{attribute 'linkalways'} 
{attribute 'no_explicit_call' := 'This FB is a CLASS and must be accessed using methods or properties'}
{attribute 'enable_dynamic_creation'}
FUNCTION_BLOCK _TcVnKeyPoint EXTENDS StructuredDatatypeBase
VAR
	localData : TcVnKeyPoint;
	activeData : REFERENCE TO TcVnKeyPoint REF= localData;
    _aPoint : _TcVnPoint2_REAL();
    _fDiameter : _REAL(localdata.fDiameter);
    _fAngle : _REAL(localdata.fAngle);
    _fResponse : _REAL(localdata.fResponse);
    _nOctave : _DINT(localdata.nOctave);
    _nClassId : _DINT(localdata.nClassId);
END_VAR

PROPERTY PUBLIC Address : PVOID
GET
Address := ADR(activeData);
END_GET
END_PROPERTY

PROPERTY PUBLIC aPoint : REFERENCE TO _TcVnPoint2_REAL
GET
aPoint REF= _aPoint;
END_GET
END_PROPERTY

METHOD PUBLIC ClearReference
VAR_INPUT
END_VAR
activeData REF= localData;
SetMemberReference();
END_METHOD

METHOD PUBLIC Clone : I_Datatype
VAR
    pClone : POINTER TO _TcVnKeyPoint;
END_VAR
pClone := __NEW(_TcVnKeyPoint());
pClone^.Value := Value;
Clone := pClone^;
END_METHOD

PROPERTY PUBLIC fAngle : REFERENCE TO _REAL
GET
fAngle REF= _fAngle;
END_GET
END_PROPERTY

METHOD FB_init : BOOL
VAR_INPUT
	bInitRetains : BOOL; // if TRUE, the retain variables are initialized (warm start / cold start)
	bInCopyCode : BOOL;  // if TRUE, the instance afterwards gets moved into the copy code (online change)
END_VAR
SetMemberReference();
AddMember('aPoint', _aPoint);
AddMember('fDiameter', _fDiameter);
AddMember('fAngle', _fAngle);
AddMember('fResponse', _fResponse);
AddMember('nOctave', _nOctave);
AddMember('nClassId', _nClassId);
END_METHOD

PROPERTY PUBLIC fDiameter : REFERENCE TO _REAL
GET
fDiameter REF= _fDiameter;
END_GET
END_PROPERTY

PROPERTY PUBLIC fResponse : REFERENCE TO _REAL
GET
fResponse REF= _fResponse;
END_GET
END_PROPERTY

PROPERTY PUBLIC Identifier : T_MAXSTRING
GET
Identifier := 'TcVnKeyPoint';
END_GET
END_PROPERTY

METHOD PUBLIC MakeReferenceTo
VAR_INPUT
	ReferenceTarget : REFERENCE TO TcVnKeyPoint;
END_VAR
activeData REF= ReferenceTarget;
SetMemberReference();
END_METHOD

PROPERTY PUBLIC nClassId : REFERENCE TO _DINT
GET
nClassId REF= _nClassId;
END_GET
END_PROPERTY

PROPERTY PUBLIC nOctave : REFERENCE TO _DINT
GET
nOctave REF= _nOctave;
END_GET
END_PROPERTY

METHOD PROTECTED SetMemberReference
VAR_INPUT
END_VAR
_aPoint.MakeReferenceTo(activeData.aPoint);
_fDiameter.MakeReferenceTo(activeData.fDiameter);
_fAngle.MakeReferenceTo(activeData.fAngle);
_fResponse.MakeReferenceTo(activeData.fResponse);
_nOctave.MakeReferenceTo(activeData.nOctave);
_nClassId.MakeReferenceTo(activeData.nClassId);
END_METHOD

PROPERTY PUBLIC Size : UDINT
GET
Size := SIZEOF(activeData);
END_GET
END_PROPERTY

METHOD TryMakeReferenceTo : BOOL
VAR_INPUT
	Target : I_Datatype;
END_VAR
VAR
	pTargetData : POINTER TO TcVnKeyPoint;
END_VAR
IF NOT IsEquivalentTo(Target) THEN
	RETURN;
END_IF

pTargetData := Target.Address;
activeData REF= pTargetData^;
SetMemberReference();
TryMakeReferenceTo := TRUE;
END_METHOD

PROPERTY PUBLIC Value : REFERENCE TO TcVnKeyPoint
GET
Value REF= activeData;
END_GET
END_PROPERTY

END_FUNCTION_BLOCK

(* stored: Version 1.1.0.1, ProductVersion 3.1.4024.13
   POU _TcVnKeyPoint: Id {4bea38db-04f4-0aed-06b6-2af97c3dac8d}, SpecialFunc None
   Folder Core: Id {cf69e9a2-8b8c-0735-2f59-6b1c8050d553}
   Folder Customize: Id {dc46dc3b-582b-0ace-0430-b3a95061c9f5}
   Folder Constructor: Id {9ae074b2-6bfb-06f1-02ad-b614ef131606}
   Folder Protected: Id {d5333aa6-e609-055c-0acd-7eb7189b6885}
   Property Address: Id {b45f8f7d-a694-055b-237d-28f00d982fce}
   Get Get: Id {5b9f4b87-aae9-0312-137f-cb889b0aa8b9}
   Property aPoint: Id {ed5d5fbe-bada-0c0c-2356-c051fc965749}
   Get Get: Id {9fcc97f2-2ef5-07c0-2c6b-12695b087f71}
   Method ClearReference: Id {faa2c625-702f-07f5-0f24-9ec3a2384cad}
   Method Clone: Id {d71dd2f7-80fd-0f86-136a-882967127783}
   Property fAngle: Id {aa2b1b7a-c6cf-0ee0-00cb-6fb4bfdfe6ed}
   Get Get: Id {40e4b50a-d680-0ec4-030a-d7eadf8aa1c2}
   Method FB_init: Id {5dae6684-1e96-0c5b-023c-935a378485bc}
   Property fDiameter: Id {bf6071fd-fadc-04af-0b8f-5074f1309d31}
   Get Get: Id {9161927b-e7aa-006f-0f77-f092328ca351}
   Property fResponse: Id {44edf430-164c-09b6-2573-3df9ae2c0ccf}
   Get Get: Id {747fc442-59bc-0dd9-013e-f8fbd1f08308}
   Property Identifier: Id {47ce8fc4-dbef-0c77-10c9-a4b393c90e74}
   Get Get: Id {00775479-2262-006c-3524-a44767f64ed1}
   Method MakeReferenceTo: Id {fd9996df-680b-05d2-357d-df524a40c753}
   Property nClassId: Id {055e93c2-db98-025c-0925-91f8c0ab525b}
   Get Get: Id {b9674b52-ad26-0f54-1dab-55eb272b3105}
   Property nOctave: Id {0a388a1b-e9d0-0125-201e-60da407ee1ee}
   Get Get: Id {2b5ae803-6f23-0a14-124b-b50f37449994}
   Method SetMemberReference: Id {ee62db05-8ea6-0771-1688-b2559198a12c}
   Property Size: Id {2726970f-adfd-03f6-0148-57da026f8829}
   Get Get: Id {ab0782f0-e039-0e01-1d61-dfba84dba83c}
   Method TryMakeReferenceTo: Id {a4dbcc93-bc72-0453-2c0b-bfcc2a572439}
   Property Value: Id {0e2fa2aa-f9f3-0c40-2db0-3d751767f514}
   Get Get: Id {553c8c11-c933-0782-24d7-71cd72b0a8dc} *)
